FUNCTION_BLOCK RemoteTrigger (* Used to trigger a control loop remotely. *)
  (* Standard: 61499-2; Description: Outputs the system time the first time the FB is triggered remotely and upon every REQ event. This FB can also be used to request the time stamp remotely. *)
  (* Version 1.0, 2017-09-05, Marc Jakobi, HTW Berlin *)
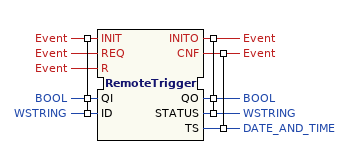
  EVENT_INPUT
    INIT WITH QI, ID; (* Initialization Request *)
    REQ; (* Service Request Event *)
    R; (* Reset Event *)
  END_EVENT
  EVENT_OUTPUT
    INITO WITH QO, STATUS; (* Initialization Confirm *)
    CNF WITH TS; (* Service Indication *)
  END_EVENT
  VAR_INPUT
    QI : BOOL; (* Input event qualifier *)
    ID : WSTRING; (* Connection identifier *)
  END_VAR
  VAR_OUTPUT
    QO : BOOL; (* Output event qualifier *)
    STATUS : WSTRING; (* Service status *)
    TS : DATE_AND_TIME; (* Time stamp *)
  END_VAR
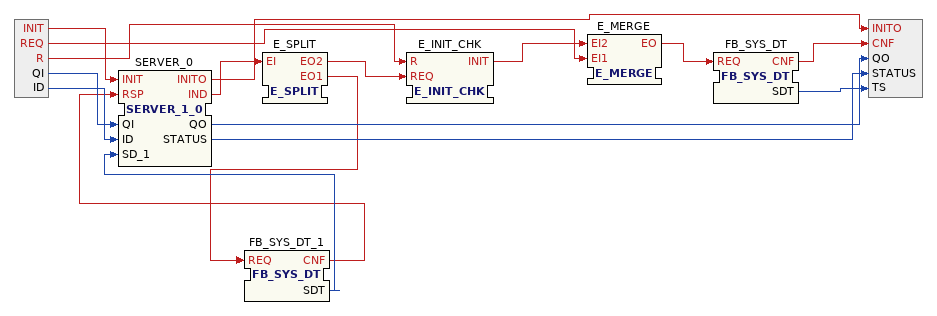
  FBS
    E_INIT_CHK : E_INIT_CHK;
    FB_SYS_DT : FB_SYS_DT;
    E_MERGE : E_MERGE;
    E_SPLIT : E_SPLIT;
    SERVER_0 : SERVER_1_0;
    FB_SYS_DT_1 : FB_SYS_DT;
  END_FBS
  EVENT_CONNECTIONS
    FB_SYS_DT.CNF TO CNF;
    E_MERGE.EO TO FB_SYS_DT.REQ;
    E_INIT_CHK.INIT TO E_MERGE.EI2;
    REQ TO E_MERGE.EI1;
    R TO E_INIT_CHK.R;
    E_SPLIT.EO2 TO E_INIT_CHK.REQ;
    INIT TO SERVER_0.INIT;
    SERVER_0.INITO TO INITO;
    SERVER_0.IND TO E_SPLIT.EI;
    E_SPLIT.EO1 TO FB_SYS_DT_1.REQ;
    FB_SYS_DT_1.CNF TO SERVER_0.RSP;
  END_CONNECTIONS
  DATA_CONNECTIONS
    FB_SYS_DT.SDT TO TS;
    QI TO SERVER_0.QI;
    ID TO SERVER_0.ID;
    SERVER_0.QO TO QO;
    SERVER_0.STATUS TO STATUS;
    FB_SYS_DT_1.SDT TO SERVER_0.SD_1;
  END_CONNECTIONS
END_FUNCTION_BLOCK
